# B&R Automation Studio project kurs
Automation Studio 4.5.2.102

## Configuration Config1

CPU 4PP065.0571-P74, AutomationRuntime D4.52, Build 4.1.2, Vc V4.52.0

### Task classes (Cpu.sw)
```
Cyclic#4:
  CRANE_1 <- CRANE_1.prg
  PLT_1 <- PLT_1.prg
Binaries: udbdef, TCData, ashwd, User, asfw, arconfig, sysconf, Role, ashwac, iomap, OpcUaMap
```

### Hardware
```
4PP065_0571_P74 : 4PP065.0571-P74 v1.1.2.0
  Connector IF5:
    ActivateDevice = 1
  ConfigurationID = kurs_Config1
  Simulation = 1
  ActivateOpcUa = 1
  OpcUa_SamplingTimer_Default = 1
  OpcUaInformationModels_PV_Version = 1
```

## Logical view

### Global.var - Global variables
```iecst
VAR
	BR_CNV : BOOL;
	go : USINT;
	crane_1_space : ARRAY[0..54] OF BOOL;
END_VAR
```

### Program Logical/PLT_1 (ANSIC)

#### Variables.var
```iecst
VAR
	BR_PLT_TURN_1 : BOOL;
	BR_PLT_SENS_1 : BOOL;
	BR_PLT_BELT_1 : BOOL;
	BR_PLT_PUSH_1 : BOOL;
	BR_PLT_PUSH_DID_1 : BOOL;
	BR_PLT_CLAMP_1 : BOOL;
	BR_PLT_CLAMP_DID_1 : BOOL;
	BR_PLT_PLATE_1 : BOOL;
	BR_PLT_PLATE_DID_1 : BOOL;
	BR_PLT_FRONT : BOOL;
	BR_PLT_BACK : BOOL;
	k : USINT;
	BR_PLT_GO : BOOL;
	BR_PLT_UP : BOOL;
	BR_PLT_CNV : BOOL;
	i : USINT;
	BR_PLT_DOWN : BOOL;
	BR_PLT_EL_FULL : BOOL;
	BR_PLT_EL_MOVING : BOOL;
END_VAR
```

#### Main.cpp
```cpp
#include <bur/plctypes.h>

#ifdef _DEFAULT_INCLUDES
	#include <AsDefault.h>
#endif

// amount of memory to be allocated for heap storage must be specified for every ANSI C++ program with the bur_heap_size variable
unsigned long bur_heap_size = 0xFFFF;

void _INIT ProgramInit(void)
{
	i=0;
	go=0;
	BR_PLT_TURN_1=1;
	BR_PLT_BELT_1=1;
	BR_CNV=1;
	BR_PLT_CNV=1;
	BR_PLT_GO=1;
	BR_PLT_UP=0;
	BR_PLT_DOWN=0;
	k=0;
	BR_PLT_EL_FULL = 1;

}

void _CYCLIC ProgramCyclic(void)
{
	if((BR_PLT_FRONT == 1) && (BR_PLT_BACK == 1) && (k==0))
	{
		BR_PLT_CNV=0;
		BR_PLT_GO=0;
		BR_PLT_EL_FULL = 1;
		BR_PLT_UP = 1;
		k++;
	}
	if((BR_PLT_EL_MOVING == 0) && (k==1))
	{
		k++;
	}
	if((BR_PLT_EL_MOVING == 1) && (k==2))
	{
		k++;
	}
	if((BR_PLT_EL_MOVING == 0) && (k==3))
	{
		BR_PLT_UP = 0;
		k++;
	}
	if(BR_PLT_SENS_1 == 1 && (i==0) && (go<2))
	{
		BR_PLT_BELT_1=1;
		BR_CNV=1;
		i++;
	}
	if((BR_PLT_SENS_1 == 0) && (i==1))
	{
		i++;
	}
	if((BR_PLT_SENS_1 == 1) && (i==2))
	{
		i++;
	}
	if((BR_PLT_SENS_1 == 0) && (i==3))
	{
		i++;
	}
	if((BR_PLT_SENS_1 == 1) && (i==4))
	{
		i++;
	}
	if((BR_PLT_SENS_1 == 0) && (i==5))
	{
		i++;
	}
	if((BR_PLT_SENS_1 == 1) && (i==6))
	{
		i++;
	}

	if(i==7)
	{
		BR_CNV=0;
		BR_PLT_BELT_1 = 0;
		i++;
	}
	while((BR_PLT_PUSH_DID_1 == 1) && (i==8))
	{
		BR_PLT_PUSH_1 = 1;
	}
	if((i==8) && (BR_PLT_PUSH_DID_1 == 0))
	{
		i++;
	}
	if((i==9) && (BR_PLT_PUSH_DID_1 == 1))
	{
		BR_PLT_PUSH_1 = 0;
		i++;
	}
	if(BR_PLT_SENS_1 == 1 && (i==10))
	{
		BR_CNV=1;
		BR_PLT_BELT_1 = 1;
		i++;
	}
	if((BR_PLT_SENS_1 == 0) && (i==11))
	{
		i++;
	}
	if((BR_PLT_SENS_1 == 1) && (i==12))
	{
		i++;
	}
	if((BR_PLT_SENS_1 == 0) && (i==13))
	{
		i++;
	}
	if((BR_PLT_SENS_1 == 1) && (i==14))
	{
		i++;
	}
	if((BR_PLT_SENS_1 == 0) && (i==15))
	{
		i++;
	}
	if((BR_PLT_SENS_1 == 1) && (i==16))
	{
		i++;
	}

	if(i==17)
	{
		BR_CNV=0;
		BR_PLT_BELT_1 = 0;
		i++;
	}
	while((BR_PLT_PUSH_DID_1 == 1) && (i==18))
	{
		BR_PLT_PUSH_1 = 1;
	}
	if((i==18) && (BR_PLT_PUSH_DID_1 == 0))
	{
		i++;
	}
	if((i==19) && (BR_PLT_PUSH_DID_1 == 1))
	{
		BR_PLT_PUSH_1 = 0;
		i++;
	}
	if((BR_PLT_PUSH_DID_1 == 1) && (i==20))
	{
		BR_PLT_CLAMP_1 = 1;
	}
	if((i==20) && (BR_PLT_CLAMP_DID_1 == 0))
	{
		i++;
	}
	if((i==21) && (BR_PLT_CLAMP_DID_1 == 1))
	{
		i++;
	}
	if((BR_PLT_PLATE_DID_1 == 1) && (i==22))
	{
		BR_PLT_PLATE_1 = 1;
		i++;
	}
	if((i==23) && (BR_PLT_PLATE_DID_1 == 0))
	{
		i++;
	}
	if((i==24) && (BR_PLT_PLATE_DID_1 == 1))
	{
		BR_PLT_EL_FULL = 0;
		BR_PLT_DOWN = 1;
		i++;
	}
	if((i==25)&&(BR_PLT_EL_MOVING == 0))
	{
		i++;
	}
	if((i==26)&&(BR_PLT_EL_MOVING == 1))
	{
		i++;
	}
	if((i==27)&&(BR_PLT_EL_MOVING == 0))
	{
		BR_PLT_CLAMP_1 = 0;
		BR_PLT_PLATE_1 = 0;
		BR_PLT_DOWN = 0;
		i=0;
		go++;
	}
	if(go==2)
	{
		BR_PLT_EL_FULL = 1;
		go++;
	}
	if(go==3)
	{
		BR_PLT_DOWN = 1;
		go++;
	}
	if((go==4)&&(BR_PLT_EL_MOVING == 1))
	{
		go++;
	}
	if((go==5)&&(BR_PLT_EL_MOVING == 0))
	{
		BR_PLT_GO = 1;
		BR_PLT_DOWN = 0;
		go++;
	}
	if((BR_PLT_FRONT == 1) && (BR_PLT_BACK == 0))
	{
		BR_PLT_CNV=1;
		k=0;
	}
}

void _EXIT ProgramExit(void)
{
	// Insert code here

}
```

### Program Logical/CRANE_1 (ANSIC)

#### Variables.var
```iecst
VAR
	BR_CRANE_SENS_1 : BOOL;
	BR_CRANE_CONV_1 : BOOL;
	i : USINT;
	BR_CRANE_TG_POS_1 : USINT;
	BR_CRANE_LIM_LEFT_1 : BOOL;
	BR_CRANE_LIM_RIGHT_1 : BOOL;
	BR_CRANE_LIM_MIDDLE_1 : BOOL;
	BR_CRANE_MOVING_X_1 : BOOL;
	BR_CRANE_MOVING_Z_1 : BOOL;
	BR_CRANE_LEFT_1 : BOOL;
	BR_CRANE_RIGHT_1 : BOOL;
	BR_CRANE_LIFT_1 : BOOL;
	n : USINT;
END_VAR
```

#### Main.c
```c
#include <bur/plctypes.h>

#ifdef _DEFAULT_INCLUDES
	#include <AsDefault.h>
#endif

void _INIT ProgramInit(void)
{
	i=0;
	n=0;
}

void _CYCLIC ProgramCyclic(void)
{
	if((go==6)&(i==0))
	{
		BR_CRANE_CONV_1 = 1;
		go=0;
		i++;
	}
	if((i==1)&&(BR_CRANE_SENS_1==1))
	{
		BR_CRANE_CONV_1 = 0;
		BR_CRANE_LEFT_1 = 1;
		i++;
	}
	if((i==2)&&(BR_CRANE_LIM_LEFT_1==1))
	{
		BR_CRANE_LIFT_1 = 1;
		i++;
	}
	if((i==3)&&(BR_CRANE_MOVING_Z_1==1))
	{
		BR_CRANE_LEFT_1 = 0;
		i++;
	}
	if((i==4)&&(BR_CRANE_LIM_MIDDLE_1==1))
	{
		while(crane_1_space[n]!=0)
		{
			n++;
		}
		crane_1_space[n] = 1;
		BR_CRANE_TG_POS_1 = (n+1);
		n=0;
		i++;
	}
	if((i==5)&&(BR_CRANE_MOVING_Z_1==1)&&(BR_CRANE_MOVING_X_1==1))
	{
		i++;
	}
	if((i==6)&&(BR_CRANE_MOVING_Z_1==0)&&(BR_CRANE_MOVING_X_1==0))
	{
		BR_CRANE_RIGHT_1 = 1;
		i++;
	}
	if((i==7)&&(BR_CRANE_LIM_RIGHT_1==1))
	{
		BR_CRANE_LIFT_1 = 0;
		i++;
	}
	if((i==8)&&(BR_CRANE_MOVING_Z_1==1))
	{
		i++;
	}
	if((i==9)&&(BR_CRANE_MOVING_Z_1==0))
	{
		BR_CRANE_RIGHT_1 = 0;
		i++;
	}
	if((i==10)&&(BR_CRANE_LIM_MIDDLE_1==1))
	{
		BR_CRANE_TG_POS_1 = 55;
		i=0;
	}
}

void _EXIT ProgramExit(void)
{

}
```

Listed in the project but not available here: Logical/Global.typ, Logical/Libraries
